FUNCTION_BLOCK FB_MatrixGetMagicSquare_Test EXTENDS FB_TestSuite
VAR_INPUT
END_VAR
VAR_OUTPUT
END_VAR
VAR
END_VAR

WhenCreatedExpectMagicProperties();

METHOD PRIVATE WhenCreatedExpectMagicProperties
VAR_INPUT
END_VAR
VAR
	M1 : DynamicMatrix;
	V : DynamicMatrix;
	Actual : LREAL;
	Expected : LREAL := 15;
	I : UINT;
END_VAR
TEST('WhenCreatedExpectMagicProperties');

// @TEST-RUN
M1.InitMagicSquare(3);//all rows and cols are 15
M1.LogData('3x3 Magic Square');

// @TEST-ASSERT
FOR I := 0 TO M1.Rows-1 DO
	//V.AsRowVector(M1,I); //cannot use, untested at this point
	Actual :=  M1.GetRC(I,0) + M1.GetRC(I,1) + M1.GetRC(I,2);//V.Sum; //cannot use, untested at this point
	AssertEquals(Expected,Actual,'Row is not the magic number');
END_FOR
FOR I := 0 TO M1.Cols-1 DO
	//V.AsRowVector(M1,I); //cannot use, untested at this point
	Actual :=  M1.GetRC(0,I) + M1.GetRC(1,I) + M1.GetRC(2,I);//V.Sum; //cannot use, untested at this point
	AssertEquals(Expected,Actual,'Col is not the magic number');
END_FOR

TEST_FINISHED();
END_METHOD

END_FUNCTION_BLOCK

(* stored: Version 1.1.0.1, ProductVersion 3.1.4024.9
   POU FB_MatrixGetMagicSquare_Test: Id {a15b73b2-380f-051b-10ff-af82c1df93a3}, SpecialFunc None
   Method WhenCreatedExpectMagicProperties: Id {8f2dca3c-5f77-06ac-0bb8-305f754aab8f} *)
